Fanuc KAREL source: tst_csv_writ.kl

PROGRAM tst_csv_writ
%NOLOCKGROUP

CONST
  WRITE_COND = 1
VAR
  csv_name FROM tst_csv_main : STRING[16]
  csv_file FROM tst_csv_main : FILE
  block_write FROM tst_csv_main : INTEGER
  waitime FROM tst_csv_main : INTEGER
  time_out : BOOLEAN

%include display.c.klt
%include systemlib.codes.klt
%include systemlib.datatypes.klt

%include display.klh
%include csv.klh

-- sensor csv file
%class tstcsv('csvclass.klc','csvclass.klh')

BEGIN
  --clear display
  display__clear
  --show display
  display__show

  WHILE(TRUE) DO
    IF tstcsv__get_lines_written >= tstcsv__get_maxlines THEN
      PEND_SEMA(block_write, waitime, time_out)

      WRITE TPDISPLAY(CR,'Flushing pipe!')

      IF time_out THEN
        GOTO ENDREAD
      ENDIF
      -- (name, file, handle open/close)
      tstcsv__write_to_file(csv_name, csv_file, TRUE)
      tstcsv__clear
      POST_SEMA(block_write)
    ENDIF
    DELAY 100
  ENDWHILE
  ENDREAD::

END tst_csv_writ
